(* CoDeSys 2.3 export: SHADERS.EXP *)

(* Global variable list: Shaders *)
VAR_GLOBAL
	shader_kuchnia:Shader;
	shader_taras:Shader;
	shader_kominek:Shader;
	shader_gabinet:Shader;
	shader_sypialnia:Shader;
	shader_lazienka:Shader;
	shader_kotlownia:Shader;
	shader_Julka:Shader;
	shader_Julka_dach:Shader;
	shader_Zosia:Shader;
	shader_Zosia_dach_L:Shader;
	shader_Zosia_dach_P:Shader;
	shader_przedpokoj:Shader;

END_VAR
